{attribute addProperty BoxType "EJ1918-0000-0017"}
{attribute addProperty Id "Module_1_FSOEModule_1_FSOE_99CFC0AE104130Module_2_DEVICEIOModule_2_DEVICEIO_FB2B67D71620Module_3_FSLOGICModule_3_FSLOGIC_3E6251391620WcStateAT %I*WcState_98A4DF7520.250InfoDataAT %I*InfoData_BC63D37F80100"}
{attribute addProperty CRC "3580821133"}
{attribute addProperty SizeInBites "218"}
{attribute addProperty SizeInBytes "27.25"}
TYPE EJ1918_151E5A82 :
STRUCT
	{attribute addProperty Name "Module_1_FSOE"}
	Module_1_FSOE : Module_1_FSOE_99CFC0AE;
	{attribute addProperty Name "Module_2_DEVICEIO"}
	Module_2_DEVICEIO : Module_2_DEVICEIO_FB2B67D7;
	{attribute addProperty Name "Module_3_FSLOGIC"}
	Module_3_FSLOGIC : Module_3_FSLOGIC_3E625139;
	{attribute addProperty Name "WcState"}
	WcState : WcState_98A4DF75;
	{attribute addProperty Name "InfoData"}
	InfoData : InfoData_BC63D37F;
END_STRUCT
END_TYPE

(* stored: Version 1.2.0.0, ProductVersion 3.1.4024.9
   DUT EJ1918_151E5A82: Id {2cf8a136-a59d-41fc-87ed-b0ed2d2abe0f} *)
